# EPICS substitutions: modules/event/evrSupport/Db/ioc/IOC-IN20-BP01evr.substitutions
#==============================================================================
#
# Abs:  LCLS EVR IOC records for IN20 BP01
#
# Name: IOC-IN20-BP01evr.substitutions
#
#==============================================================================
#
file evrBPXX.db
{
pattern { DEVICE        }
	{ EVR:IN20:BP01 }
}
